{attribute 'qualified_only'}
VAR_GLOBAL
	test: BOOL;
END_VAR

(* stored: Version 1.1.0.1, ProductVersion 3.1.4024.11
   GVL DataProces: Id {0d5a7b02-a7d8-4892-97ec-058d0980cf0f} *)
